FUNCTION_BLOCK T_ManualMode IMPLEMENTS I_PackMLMode
VAR
	
END_VAR

END_FUNCTION_BLOCK

(* stored: Version 1.1.0.1, ProductVersion 3.1.4024.12
   POU T_ManualMode: Id {339991d4-876f-4668-acda-cc2d207d93a2}, SpecialFunc None *)
